// TIA Portal V20 export
FUNCTION "LER_PartData_VisionPos" : Void   // FC10001, LAD
// stored: Access Published, SetENOAutomatically false
   VAR_INPUT
      generateCondition : Bool;
      specialFunctions : "LAF_typeSpecialFunctions";
      gaugeRnR_Type1Count : "LER_typeCount";
      gaugeRnR_Type3Count : "LER_typeCount";
      gaugeRnR_Type3PartsCount : "LER_typeCount";
      PartOn : Bool;
      JudgmentOK : Bool;
      JudgmentNG : Bool;
      JudgmentBusy : Bool;
      VisionData : "LER_typeVisionResultData";
   END_VAR
   VAR_OUTPUT
      PartData : "LER_typePartData";
   END_VAR
   VAR_TEMP
      tempRET_VAL : Word;
   END_VAR
   VAR CONSTANT
      PartStatus_Busy : Byte := 16#2;
      PartStatus_Ok : Byte := 16#3;
      PartStatus_NG : Byte := 16#4;
      TRUE : Bool := TRUE;
   END_VAR
   VAR_TEMP   // added for the SCL form of the ladder/FBD networks
      _w1 : Bool;
      _w2 : Bool;
   END_VAR
BEGIN

REGION Network 1: ************* Nomal Mode ****************
END_REGION

REGION Network 2: PartStatus
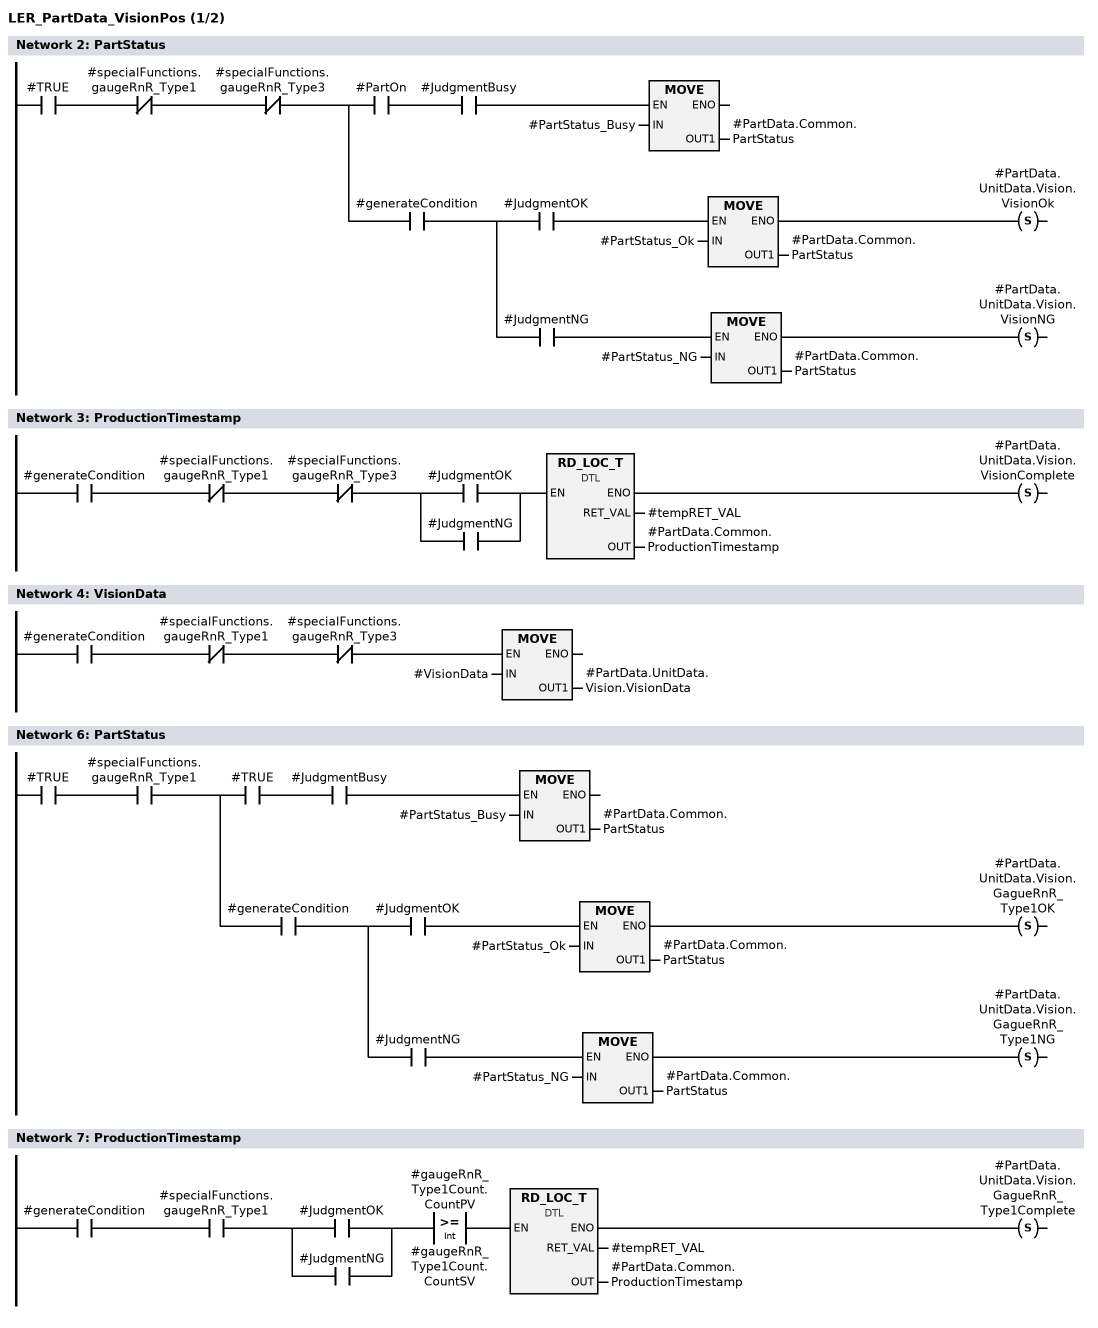
   RUNG wire#powerrail
      Contact( #TRUE )
      I_Contact( #specialFunctions.gaugeRnR_Type1 )
      I_Contact( #specialFunctions.gaugeRnR_Type3 )
      wire#w1
      Contact( #PartOn )
      Contact( #JudgmentBusy )
      Move(in := #PartStatus_Busy, out1 => #PartData.Common.PartStatus)
   END_RUNG
   RUNG wire#w1
      Contact( #generateCondition )
      wire#w2
      Contact( #JudgmentOK )
      Move(in := #PartStatus_Ok, out1 => #PartData.Common.PartStatus)
      S_Coil( #PartData.UnitData.Vision.VisionOk )
   END_RUNG
   RUNG wire#w2
      Contact( #JudgmentNG )
      Move(in := #PartStatus_NG, out1 => #PartData.Common.PartStatus)
      S_Coil( #PartData.UnitData.Vision.VisionNG )
   END_RUNG
   // the same network as SCL:
   #_w1 := #TRUE AND NOT #specialFunctions.gaugeRnR_Type1 AND NOT #specialFunctions.gaugeRnR_Type3;
   IF #_w1 AND #PartOn AND #JudgmentBusy THEN #PartData.Common.PartStatus := #PartStatus_Busy; END_IF;
   #_w2 := #_w1 AND #generateCondition;
   IF #_w2 AND #JudgmentOK THEN
       #PartData.Common.PartStatus := #PartStatus_Ok;
       #PartData.UnitData.Vision.VisionOk := TRUE;
   END_IF;
   IF #_w2 AND #JudgmentNG THEN
       #PartData.Common.PartStatus := #PartStatus_NG;
       #PartData.UnitData.Vision.VisionNG := TRUE;
   END_IF;
END_REGION

REGION Network 3: ProductionTimestamp
   RUNG wire#powerrail
      Contact( #generateCondition )
      I_Contact( #specialFunctions.gaugeRnR_Type1 )
      I_Contact( #specialFunctions.gaugeRnR_Type3 )
      wire#w1
      Contact( #JudgmentOK )
      wire#w2
      { S7_Templates := "date_type := DTL" } RD_LOC_T(RET_VAL => #tempRET_VAL, OUT => #PartData.Common.ProductionTimestamp)
      S_Coil( #PartData.UnitData.Vision.VisionComplete )
   END_RUNG
   RUNG wire#w1
      Contact( #JudgmentNG )
   END_RUNG wire#w2
   // the same network as SCL:
   #tempRET_VAL := RD_LOC_T(EN := #generateCondition AND NOT #specialFunctions.gaugeRnR_Type1 AND NOT #specialFunctions.gaugeRnR_Type3 AND (#JudgmentOK OR #JudgmentNG),
                           OUT => #PartData.Common.ProductionTimestamp,
                           ENO => #_w1);
   IF #_w1 THEN #PartData.UnitData.Vision.VisionComplete := TRUE; END_IF;
END_REGION

REGION Network 4: VisionData
   RUNG wire#powerrail
      Contact( #generateCondition )
      I_Contact( #specialFunctions.gaugeRnR_Type1 )
      I_Contact( #specialFunctions.gaugeRnR_Type3 )
      Move(in := #VisionData, out1 => #PartData.UnitData.Vision.VisionData)
   END_RUNG
   // the same network as SCL:
   IF #generateCondition AND NOT #specialFunctions.gaugeRnR_Type1 AND NOT #specialFunctions.gaugeRnR_Type3 THEN
       #PartData.UnitData.Vision.VisionData := #VisionData;
   END_IF;
END_REGION

REGION Network 5: ************* GaugeR&rType1 ****************
END_REGION

REGION Network 6: PartStatus
   RUNG wire#powerrail
      Contact( #TRUE )
      Contact( #specialFunctions.gaugeRnR_Type1 )
      wire#w1
      Contact( #TRUE )
      Contact( #JudgmentBusy )
      Move(in := #PartStatus_Busy, out1 => #PartData.Common.PartStatus)
   END_RUNG
   RUNG wire#w1
      Contact( #generateCondition )
      wire#w2
      Contact( #JudgmentOK )
      Move(in := #PartStatus_Ok, out1 => #PartData.Common.PartStatus)
      S_Coil( #PartData.UnitData.Vision.GagueRnR_Type1OK )
   END_RUNG
   RUNG wire#w2
      Contact( #JudgmentNG )
      Move(in := #PartStatus_NG, out1 => #PartData.Common.PartStatus)
      S_Coil( #PartData.UnitData.Vision.GagueRnR_Type1NG )
   END_RUNG
   // the same network as SCL:
   #_w1 := #TRUE AND #specialFunctions.gaugeRnR_Type1;
   IF #_w1 AND #TRUE AND #JudgmentBusy THEN #PartData.Common.PartStatus := #PartStatus_Busy; END_IF;
   #_w2 := #_w1 AND #generateCondition;
   IF #_w2 AND #JudgmentOK THEN
       #PartData.Common.PartStatus := #PartStatus_Ok;
       #PartData.UnitData.Vision.GagueRnR_Type1OK := TRUE;
   END_IF;
   IF #_w2 AND #JudgmentNG THEN
       #PartData.Common.PartStatus := #PartStatus_NG;
       #PartData.UnitData.Vision.GagueRnR_Type1NG := TRUE;
   END_IF;
END_REGION

REGION Network 7: ProductionTimestamp
   RUNG wire#powerrail
      Contact( #generateCondition )
      Contact( #specialFunctions.gaugeRnR_Type1 )
      wire#w1
      Contact( #JudgmentOK )
      wire#w2
      { S7_Templates := "SrcType := Int" } GE_Contact(in1 := #gaugeRnR_Type1Count.CountPV, in2 := #gaugeRnR_Type1Count.CountSV)
      { S7_Templates := "date_type := DTL" } RD_LOC_T(RET_VAL => #tempRET_VAL, OUT => #PartData.Common.ProductionTimestamp)
      S_Coil( #PartData.UnitData.Vision.GagueRnR_Type1Complete )
   END_RUNG
   RUNG wire#w1
      Contact( #JudgmentNG )
   END_RUNG wire#w2
   // the same network as SCL:
   #tempRET_VAL := RD_LOC_T(EN := #generateCondition AND #specialFunctions.gaugeRnR_Type1 AND (#JudgmentOK OR #JudgmentNG) AND (#gaugeRnR_Type1Count.CountPV >= #gaugeRnR_Type1Count.CountSV),
                           OUT => #PartData.Common.ProductionTimestamp,
                           ENO => #_w1);
   IF #_w1 THEN #PartData.UnitData.Vision.GagueRnR_Type1Complete := TRUE; END_IF;
END_REGION

REGION Network 8: VisionData
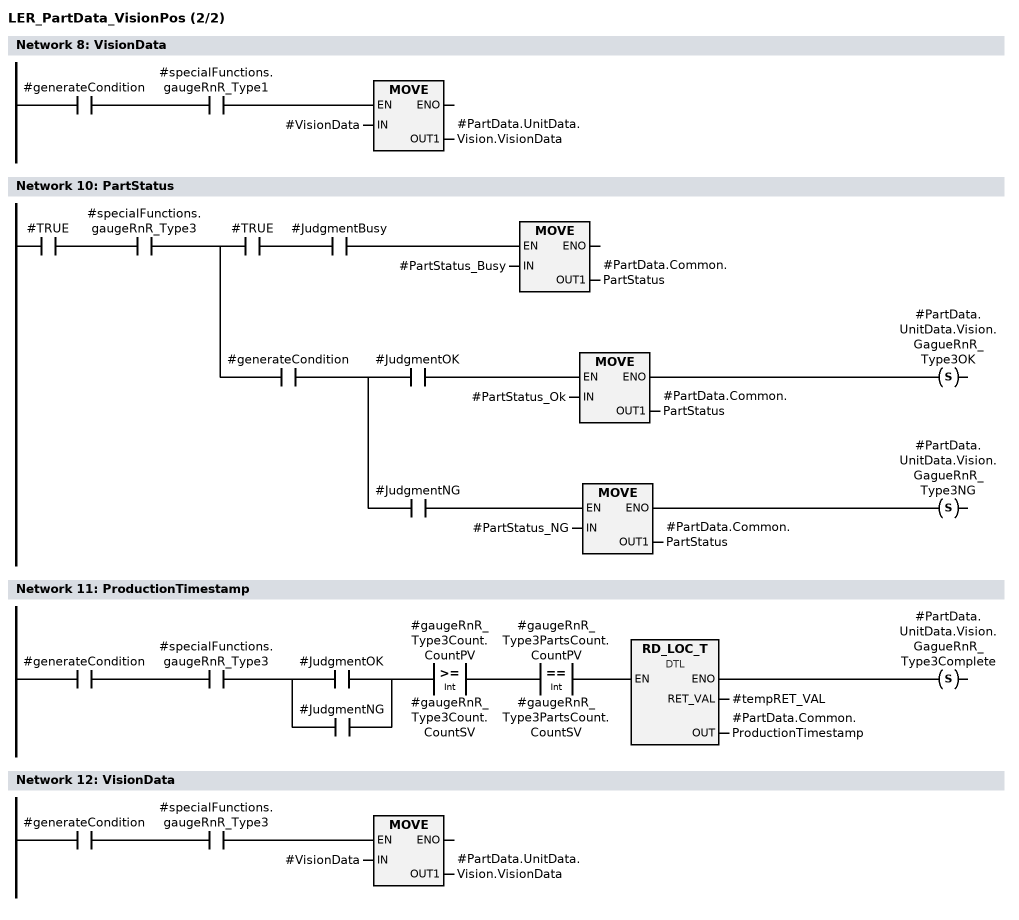
   RUNG wire#powerrail
      Contact( #generateCondition )
      Contact( #specialFunctions.gaugeRnR_Type1 )
      Move(in := #VisionData, out1 => #PartData.UnitData.Vision.VisionData)
   END_RUNG
   // the same network as SCL:
   IF #generateCondition AND #specialFunctions.gaugeRnR_Type1 THEN
       #PartData.UnitData.Vision.VisionData := #VisionData;
   END_IF;
END_REGION

REGION Network 9: ************* GaugeR&rType3 ****************
END_REGION

REGION Network 10: PartStatus
   RUNG wire#powerrail
      Contact( #TRUE )
      Contact( #specialFunctions.gaugeRnR_Type3 )
      wire#w1
      Contact( #TRUE )
      Contact( #JudgmentBusy )
      Move(in := #PartStatus_Busy, out1 => #PartData.Common.PartStatus)
   END_RUNG
   RUNG wire#w1
      Contact( #generateCondition )
      wire#w2
      Contact( #JudgmentOK )
      Move(in := #PartStatus_Ok, out1 => #PartData.Common.PartStatus)
      S_Coil( #PartData.UnitData.Vision.GagueRnR_Type3OK )
   END_RUNG
   RUNG wire#w2
      Contact( #JudgmentNG )
      Move(in := #PartStatus_NG, out1 => #PartData.Common.PartStatus)
      S_Coil( #PartData.UnitData.Vision.GagueRnR_Type3NG )
   END_RUNG
   // the same network as SCL:
   #_w1 := #TRUE AND #specialFunctions.gaugeRnR_Type3;
   IF #_w1 AND #TRUE AND #JudgmentBusy THEN #PartData.Common.PartStatus := #PartStatus_Busy; END_IF;
   #_w2 := #_w1 AND #generateCondition;
   IF #_w2 AND #JudgmentOK THEN
       #PartData.Common.PartStatus := #PartStatus_Ok;
       #PartData.UnitData.Vision.GagueRnR_Type3OK := TRUE;
   END_IF;
   IF #_w2 AND #JudgmentNG THEN
       #PartData.Common.PartStatus := #PartStatus_NG;
       #PartData.UnitData.Vision.GagueRnR_Type3NG := TRUE;
   END_IF;
END_REGION

REGION Network 11: ProductionTimestamp
   RUNG wire#powerrail
      Contact( #generateCondition )
      Contact( #specialFunctions.gaugeRnR_Type3 )
      wire#w1
      Contact( #JudgmentOK )
      wire#w2
      { S7_Templates := "SrcType := Int" } GE_Contact(in1 := #gaugeRnR_Type3Count.CountPV, in2 := #gaugeRnR_Type3Count.CountSV)
      { S7_Templates := "SrcType := Int" } EQ_Contact(in1 := #gaugeRnR_Type3PartsCount.CountPV, in2 := #gaugeRnR_Type3PartsCount.CountSV)
      { S7_Templates := "date_type := DTL" } RD_LOC_T(RET_VAL => #tempRET_VAL, OUT => #PartData.Common.ProductionTimestamp)
      S_Coil( #PartData.UnitData.Vision.GagueRnR_Type3Complete )
   END_RUNG
   RUNG wire#w1
      Contact( #JudgmentNG )
   END_RUNG wire#w2
   // the same network as SCL:
   #tempRET_VAL := RD_LOC_T(EN := #generateCondition AND #specialFunctions.gaugeRnR_Type3 AND (#JudgmentOK OR #JudgmentNG) AND (#gaugeRnR_Type3Count.CountPV >= #gaugeRnR_Type3Count.CountSV) AND (#gaugeRnR_Type3PartsCount.CountPV = #gaugeRnR_Type3PartsCount.CountSV),
                           OUT => #PartData.Common.ProductionTimestamp,
                           ENO => #_w1);
   IF #_w1 THEN #PartData.UnitData.Vision.GagueRnR_Type3Complete := TRUE; END_IF;
END_REGION

REGION Network 12: VisionData
   RUNG wire#powerrail
      Contact( #generateCondition )
      Contact( #specialFunctions.gaugeRnR_Type3 )
      Move(in := #VisionData, out1 => #PartData.UnitData.Vision.VisionData)
   END_RUNG
   // the same network as SCL:
   IF #generateCondition AND #specialFunctions.gaugeRnR_Type3 THEN
       #PartData.UnitData.Vision.VisionData := #VisionData;
   END_IF;
END_REGION
END_FUNCTION
